Fanuc KAREL source: kf00117.KL

-- PROVISIONAL review KL for V770-1; original PC SHA256 7c924cf1daab1069d7d8296b3178a5e6a9b4c65c404f1fd2e954c39383bcb18a
-- Incomplete behavior may be omitted. Consult companion uncertainty JSON. Do not deploy.
PROGRAM KF00117
%NOLOCKGROUP
BEGIN
  -- UNRESOLVED_PC offsets 0-1; opcodes 7B
  -- UNRESOLVED_PC offsets 6-21; opcodes 17,9D,33,34,23
  -- UNRESOLVED_PC offsets 26-30; opcodes 7F
  -- UNRESOLVED_PC offsets 35-45; opcodes 27,22,AA
  -- UNRESOLVED_PC offsets 50-54; opcodes 7F
END KF00117
